INTERFACE I_AssertResult

METHOD PUBLIC ReportResult
VAR_INPUT
    Expected : ANY;
    Actual : ANY;
    sMessage : Tc2_System.T_MaxString;
    sTestInstancePath : Tc2_System.T_MaxString;
END_VAR
VAR_OUTPUT
    bAlreadyReported : BOOL := FALSE;
END_VAR
END_METHOD

END_INTERFACE

(* stored: Version 1.1.0.1, ProductVersion 3.1.4022.12
   Itf I_AssertResult: Id {ed69e1f9-422b-49c9-b13a-a9f6e70684df}
   Method ReportResult: Id {9ccb96c6-63d5-4241-a84a-687a6d2fb91a} *)
